// TIA Portal V19 export
DATA_BLOCK "DecoilersHRot_PERS"   // DB68
// stored: MemoryReserve 100
   VAR RETAIN
      PersistentValues : Struct
         Par : Struct
            TraslationAx : "Positioning_DOL_Machine_Par";
            TraslationEnc : "PosFbk_RTN";
            Traslation_AutSpeed : Real := 0.0;
         END_STRUCT;
         Ax_Pers { ExternalAccessible := 'False'; ExternalVisible := 'False'; ExternalWritable := 'False'} : "Positioning_DOL_Machine_Pers_Data";
      END_STRUCT;
   END_VAR
BEGIN
   PersistentValues.Par.TraslationAx.PosTolerance := 0.1;
   PersistentValues.Par.TraslationAx.Minus_Limit := 74.0;
   PersistentValues.Par.TraslationAx.Plus_Limit := 230.0;
   PersistentValues.Par.TraslationAx.PreCutOff := 0.1;
   PersistentValues.Par.TraslationAx.PreEndLowSpeed := 2.0;
   PersistentValues.Par.TraslationAx.PreEndMedSpeed := 5.0;
   PersistentValues.Par.TraslationAx.LowSpeed := 41.0;
   PersistentValues.Par.TraslationAx.MedSpeed := 70.0;
   PersistentValues.Par.TraslationAx.HighSpeed := 70.0;
   PersistentValues.Par.TraslationAx.Man_Speed := 100.0;
   PersistentValues.Par.TraslationEnc.Preset.Pulses := -1_018_197_168;
   PersistentValues.Par.TraslationEnc.Preset.Units := 110.0;
   PersistentValues.Par.TraslationEnc.Config.Resolution := 8.0;
   PersistentValues.Ax_Pers.AxisHomed := TRUE;
END_DATA_BLOCK
